FUNCTION_BLOCK DynamicStringBuffer_TEST EXTENDS FB_TestSuite

LogsManyMessagesForManyCycles();

METHOD LogsManyMessagesForManyCycles
VAR
	result : STRING := '';
	expected : STRING := '';
	i : UDINT;
END_VAR
VAR CONSTANT
	Cycles : UDINT := 50;
	Messages : UDINT := 50;
END_VAR
VAR_INST
	cycleCount : UDINT := 0;
	logsManyMessagesForManyCyclesLogger : TcLogCore(BufferSize:=50 * 50 * 280); // Cycles * Messages * (max string length + fifo overhead (estimated))
	logger : TcLog;
END_VAR
TEST('LogsManyMessagesForManyCycles');

logsManyMessagesForManyCyclesLogger
	.WriteToFile('c:\UnitTest\', 'test.txt')
	.RunLogger();
logger.SetLogger(logsManyMessagesForManyCyclesLogger);

IF cycleCount < Cycles THEN
	FOR i:=0 TO Messages DO
		logger
			.AppendString('Cycle: ')
			.AppendString(UDINT_TO_STRING(cycleCount))
			.AppendString(', Message: ')
			.AppendString(UDINT_TO_STRING(i))
			.Error('');	
	END_FOR
END_IF
cycleCount := cycleCount + 1;

// Catch any occuring error message
IF LEN(logsManyMessagesForManyCyclesLogger.Error.Info) > 0 THEN
	result := logsManyMessagesForManyCyclesLogger.Error.Info;
END_IF

IF cycleCount > (Cycles * Messages * 2 + 4) THEN 
	AssertEquals(Expected := expected,
				 Actual := result,
				 Message := result);
 
	TEST_FINISHED();
END_IF
END_METHOD

END_FUNCTION_BLOCK

(* stored: Version 1.1.0.1
   POU DynamicStringBuffer_TEST: Id {03045c1a-5281-4fe3-bc16-4d9ce12d6b50}, SpecialFunc None
   Method LogsManyMessagesForManyCycles: Id {e452a053-adba-401f-a1d2-1bba967ad2c0} *)
